// TIA Portal V20 export
ORGANIZATION_BLOCK "DiagnosticErrorInterrupt"   // OB82, LAD, DiagnosticErrorInterrupt
// stored: SetENOAutomatically false
   VAR_INPUT
      IO_State : Word;   // IO state of the HW object
      LADDR : HW_ANY;   // Hardware identifier
      Channel : UInt;   // Channel number
      MultiError : Bool;   // =true if more than one error is present
   END_VAR
BEGIN
END_ORGANIZATION_BLOCK
